FUNCTION_BLOCK AB5Policy
  (* Standard: 61499-2 *)
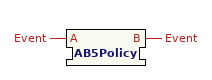
  EVENT_INPUT
    A;
  END_EVENT
  EVENT_OUTPUT
    B;
  END_EVENT
END_FUNCTION_BLOCK
(* other elements stored in the file *)
(* Name  AB5 *)
(* VarDeclaration Name=v Type=dtimer *)
(* Name  s0 *)
(* Name  s1 *)
(* ECTransition Source=s0 Destination=s0 Condition=( !A and !B ) *)
(* VarName  v *)
(* Value  0 *)
(* ECTransition Source=s0 Destination=s1 Condition=( A and !B ) *)
(* VarName  v *)
(* Value  0 *)
(* ECTransition Source=s0 Destination=violation Condition=( ( !A and B ) or ( A and B ) ) *)
(* ECTransition Source=s1 Destination=s1 Condition=( !A and !B and v < 5 ) *)
(* ECTransition Source=s1 Destination=s0 Condition=( !A and B ) *)
(* ECTransition Source=s1 Destination=violation Condition=( ( v >= 5 ) or ( A and B ) or ( A and !B ) ) *)
